(* IEC 61131-3 sources: POMIRTS_lab3/AS/Library/AsSound, 2 files *)

(* ---- AsSound.fun ---- *)
(********************************************************************
 * COPYRIGHT -- Bernecker + Rainer
 ********************************************************************
 * Library: AsSound
 * File: AsSound.fun
 * Author: B+R
 ********************************************************************
 * Functions and function blocks of library AsSound
 ********************************************************************)

FUNCTION_BLOCK sndCreateSound			(*SND - create a sndObj*)
	VAR_INPUT
		enable			: BOOL;			(*enables execution*)
		pDevice			: UDINT;		(*Devicename given as a pointer*)
		pFile			: UDINT;		(*Filename given as a pointer*)
	END_VAR

	VAR_OUTPUT
		status			: UINT;			(*execution status: ERR_OK, ERR_FUB_ENABLE_FALSE, ERR_FUB_BUSY, 0xXXXX = see help*)
		hSound			: UDINT;		(*handle of sndObj*)
	END_VAR

	VAR
        i_state			: UINT;			(*internal variable*)
		i_result		: UINT;			(*internal variable*)
        i_tmp			: UDINT;		(*internal variable*)
	END_VAR
END_FUNCTION_BLOCK

FUNCTION_BLOCK sndCtrlSound				(*SND - control a sndObj*)
	VAR_INPUT
		enable			: BOOL;			(*enables execution*)
		hSound			: UDINT;		(*Handle of sndObj*)
		fSound			: UDINT;		(*controlling flag*)
	END_VAR

	VAR_OUTPUT
		status			: UINT;			(*execution status: ERR_OK, ERR_FUB_ENABLE_FALSE, ERR_FUB_BUSY, 0xXXXX = see help*)
	END_VAR

	VAR
        i_state			: UINT;			(*internal variable*)
		i_result		: UINT;			(*internal variable*)
        i_tmp			: UDINT;		(*internal variable*)
	END_VAR
END_FUNCTION_BLOCK

FUNCTION sndSetVolume : UINT 			(*SND - change volume level*)
	VAR_INPUT
		volumeLevel	: USINT;			(*volume level [0,100]*)
	END_VAR
END_FUNCTION

FUNCTION sndSetMute : UINT 				(*SND - mute on/off*)
	VAR_INPUT
		muteSwitch	: USINT;			(*mute switch [0,1]*)
	END_VAR
END_FUNCTION

(* ---- AsSound.var ---- *)
(********************************************************************
 * COPYRIGHT -- Bernecker + Rainer
 ********************************************************************
 * Library: AsSound
 * File: AsSound.var
 * Author: B+R
 ********************************************************************
 * Local variables of library AsSound
 ********************************************************************)

VAR CONSTANT
	sndERR_NODRIVER				: UINT		:= 35050;	(*no device driver is present*)
	sndERR_INVALID_PARAM		: UINT		:= 35051;	(*invalid parameters*)
	sndERR_FILE_NOT_FOUND		: UINT		:= 35052;	(*file not found*)
	sndERR_ALLOCATED			: UINT		:= 35053;	(*specified resource is already allocated*)
	sndERR_BAD_FORMAT			: UINT		:= 35054;	(*attempted to open with an unsupported waveform-audio format*)
	sndERR_NOMEM				: UINT		:= 35055;	(*unable to allocate or lock memory*)
	sndERR_LIMIT_STREAMS		: UINT		:= 35056;	(*maximum number of playback streams reached*)
	sndERR_MODE_EXCLUSIVE		: UINT		:= 35057;	(*exclusive more enabled for a deddicated snd-object*)
	sndERR_OUT_OF_RANGE			: UINT		:= 35058;	(*volume level out of range [0,100]*)

	sndDELETE					: UINT		:= 1;		(*delete snd-object*)
	sndSTOP						: UINT		:= 2;		(*stop snd-object*)
	sndPLAY						: UINT		:= 3;		(*play snd-object*)
	sndPAUSE					: UINT		:= 4;		(*pause snd-object*)

	sndEXCLUSIVE				: UINT		:= 16;		(*exclusive playback*)
	sndLOOP						: UINT		:= 32;		(*loop playback*)
END_VAR
